{attribute 'GeneratedUsingTerminal: EL5072-0000-0016'}
{attribute addProperty BoxType "EL5072-0000-0016"}
{attribute addProperty Id "EtcSlaveTerminalBaseIND_Inputs_Channel_1AT %I*IND_Inputs_Channel_BBE8401F18IND_Inputs_Channel_2AT %I*IND_Inputs_Channel_BBE8401F18IND_Outputs_Channel_1AT %Q*IND_Outputs_Channel_02FDE6C97IND_Outputs_Channel_2AT %Q*IND_Outputs_Channel_02FDE6C97WcStateAT %I*WcState_9091E0EB2InfoDataAT %I*InfoData_32EB74EA10"}
{attribute addProperty CRC "2114576108"}
{attribute addProperty Size "62"}
TYPE EL5072_7E09DEEC EXTENDS EtcSlaveTerminalBase :
STRUCT
	{attribute addProperty Name "IND_Inputs_Channel_1"}
	IND_Inputs_Channel_1 : IND_Inputs_Channel_BBE8401F;
	{attribute addProperty Name "IND_Inputs_Channel_2"}
	IND_Inputs_Channel_2 : IND_Inputs_Channel_BBE8401F;
	{attribute addProperty Name "IND_Outputs_Channel_1"}
	IND_Outputs_Channel_1 : IND_Outputs_Channel_02FDE6C9;
	{attribute addProperty Name "IND_Outputs_Channel_2"}
	IND_Outputs_Channel_2 : IND_Outputs_Channel_02FDE6C9;
	{attribute addProperty Name "WcState"}
	WcState : WcState_9091E0EB;
	{attribute addProperty Name "InfoData"}
	InfoData : InfoData_32EB74EA;
END_STRUCT
END_TYPE

(* stored: Version 1.2.0.0, ProductVersion 3.1.4024.9
   DUT EL5072_7E09DEEC: Id {ff51166d-8d27-4d0e-8237-959c20ea9e52} *)
